{attribute 'GeneratedUsingTerminal: EL4011-0000-0016'}
{attribute addProperty BoxType "EL4011-0000-0016"}
{attribute addProperty Id "EtcSlaveTerminalBaseAO_OutputsAT %Q*AO_Outputs_BA7EBB7C2WcStateAT %I*WcState_0B2B16F91InfoDataAT %I*InfoData_32EB74EA10"}
{attribute addProperty CRC "1880743030"}
{attribute addProperty Size "13"}
TYPE EL4011_7019DC76 EXTENDS EtcSlaveTerminalBase :
STRUCT
	{attribute addProperty Name "AO_Outputs"}
	AO_Outputs : AO_Outputs_BA7EBB7C;
	{attribute addProperty Name "WcState"}
	WcState : WcState_0B2B16F9;
	{attribute addProperty Name "InfoData"}
	InfoData : InfoData_32EB74EA;
END_STRUCT
END_TYPE

(* stored: Version 1.2.0.0, ProductVersion 3.1.4024.9
   DUT EL4011_7019DC76: Id {9434e95f-6e97-4b10-ae0e-736129a1010d} *)
